PROGRAM FEED
VAR
END_VAR

END_PROGRAM

(* stored: Version 1.1.0.1, ProductVersion 3.1.4024.12
   POU FEED: Id {5ff3d1d0-210e-41a5-9143-c2f89242d313}, SpecialFunc None *)
